FUNCTION_BLOCK EL2788
VAR
	{attribute addProperty Name "WcState"}
	_wcState : WcStateBase;
	{attribute addProperty Name "Info data"}
	_infoData : InfoDataBase;
	_io : EL2xx8_Data;
END_VAR

PROPERTY IO : REFERENCE TO EL2xx8_Data
GET
IO REF= _io;
END_GET
END_PROPERTY

PROPERTY WcState : REFERENCE TO WcStateBase
GET
WcState REF= _wcState;
END_GET
END_PROPERTY

END_FUNCTION_BLOCK

(* stored: Version 1.1.0.1, ProductVersion 3.1.4024.9
   POU EL2788: Id {7c08a6fd-197b-09d0-0468-1b1f4f4725d8}, SpecialFunc None
   Property IO: Id {9504a29b-6956-0f7b-2d50-e8eef47ec0b8}
   Get Get: Id {0d8d2128-3fd6-0a8f-31d4-5d6415ac42f6}
   Property WcState: Id {3897ed16-7ee8-0099-3c36-7d064c2f1f85}
   Get Get: Id {c445be94-c288-062a-19a6-4e0eace7f27a} *)
